RoboDK station: ur5_and_table_and_gripper.rdk

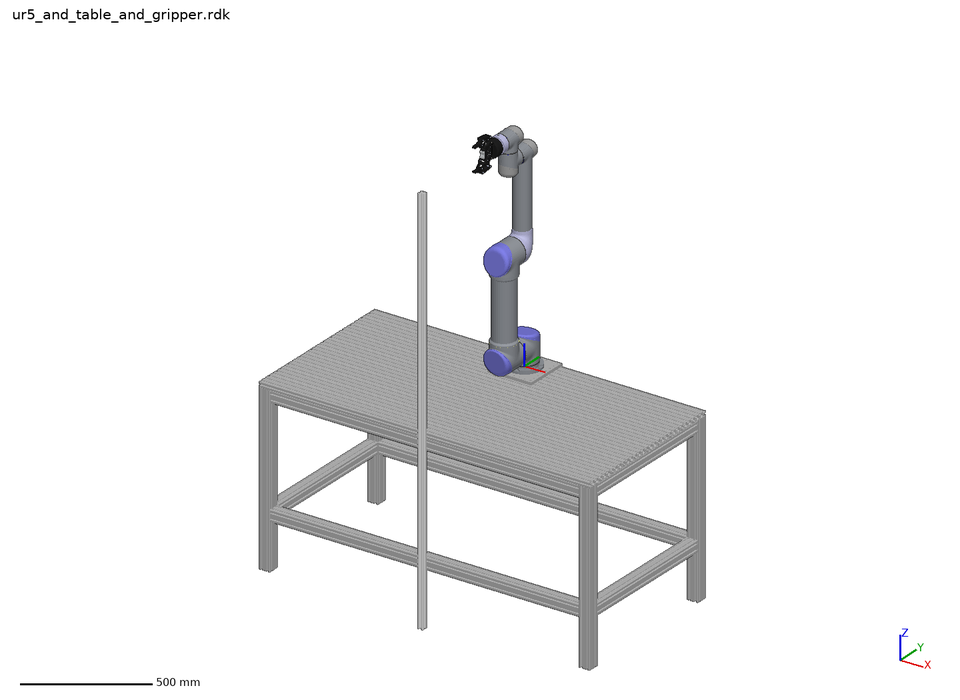
[picture v0: the station drawn from its stored meshes, robots at their saved joint values, targets as dots, program paths as lines]
Station ur5_and_table_and_gripper (saved by RoboDK 5.3.4). Poses are relative to the parent item; angles as X-Y-Z fixed-axis rotations.
  - frame UR5 Base at (0, 0, 0) mm
    - robot UR5: 6 axes, payload 5 kg, reach 850 mm, repeatability 0.1 mm, weight 18.4 kg
        modified DH rows (alpha deg, a mm, theta deg, d mm): 0, 0, 0, 89.2; 90, 0, 180, 0; 0, 425, 0, 0; 0, 392.43, 0, 109; -90, 0, 0, 93.65; 90, 0, 180, 82
        joint limits [-360, -360, -360, -360, -360, -360] to [360, 360, 360, 360, 360, 360]; home [0, -90, 90, 0, 90, 0]; saved at [0, -90, 0, -90, 0, 0]
      - tool Gripper RobotiQ 85 Opened, TCP at (0, 0, 149.6) mm, size 147.4 x 146.8 x 75 mm
  - object table_base_setup at (0, 0, 0) mm, rotated rx 0 ry 0 rz -90 deg, size 1524 x 762 x 800.1 mm, geometry from table_base_setup.STEP
  - object 6ft_beam_table at (0, -675, 1000) mm, size 25.4 x 25.4 x 1828.8 mm, geometry from 6ft_beam_table.IGS
  - Python program Task1 (listed below)
  - Python program Task 2 (listed below)
  - Python program Task 3 (listed below)

--- Python program Task1 ---
# This macro shows an example of running a program on the robot using the Python API (online programming)
# More information about the RoboDK API appears here:
# https://robodk.com/doc/en/RoboDK-API.html
from robolink import *    # API to communicate with RoboDK
from robodk import *      # robodk robotics toolbox
# Any interaction with RoboDK must be done through RDK:
RDK = Robolink()
# Select a robot (a popup is displayed if more than one robot is available)
robot = RDK.ItemUserPick('Select a robot', ITEM_TYPE_ROBOT)
if not robot.Valid():
    raise Exception('No robot selected or available')
RUN_ON_ROBOT = False
# Important: by default, the run mode is RUNMODE_SIMULATE
# If the program is generated offline manually the runmode will be RUNMODE_MAKE_ROBOTPROG,
# Therefore, we should not run the program on the robot
if RDK.RunMode() != RUNMODE_SIMULATE:
    RUN_ON_ROBOT = False
if RUN_ON_ROBOT:

    # Connect to the robot using default IP
    success = robot.Connect() # Try to connect once
    status, status_msg = robot.ConnectedState()
    if status != ROBOTCOM_READY:
        # Stop if the connection did not succeed
        print(status_msg)
        raise Exception("Failed to connect: " + status_msg)
    # This will set to run the API programs on the robot and the simulator (online programming)
    RDK.setRunMode(RUNMODE_RUN_ROBOT)



# Get the current joint position of the robot
# (updates the position on the robot simulator)
joints_ref = robot.Joints()
# get the current position of the TCP with respect to the reference frame:
# (4x4 matrix representing position and orientation)
target_ref = robot.Pose()
pos_ref = target_ref.Pos()
# It is important to provide the reference frame and the tool frames when generating programs offline
# It is important to update the TCP on the robot mostly when using the driver
robot.setPoseFrame(robot.PoseFrame())
robot.setPoseTool(robot.PoseTool())
#robot.setZoneData(10) # Set the rounding parameter (Also known as: CNT, APO/C_DIS, ZoneData, Blending radius, cornering, ...)





#Header above is re-used from the file provided for the first lab, not sure if all of it is needed but it can't hurt

#Actual Task 1 RoboDK Python segment:

#run rq_open
robot.RunCodeCustom('rq_open()',INSTRUCTION_CALL_PROGRAM)
robot.RunCodeCustom('sleep(5)',INSTRUCTION_CALL_PROGRAM)
#run rq_close
robot.RunCodeCustom('rq_close()',INSTRUCTION_CALL_PROGRAM)
robot.RunCodeCustom('sleep(5)',INSTRUCTION_CALL_PROGRAM)
#run rq_open_and_wait()
robot.RunCodeCustom('rq_open_and_wait()',INSTRUCTION_CALL_PROGRAM)
robot.RunCodeCustom('sleep(5)',INSTRUCTION_CALL_PROGRAM)
#run rq_close_and_wait()
robot.RunCodeCustom('rq_close_and_wait()',INSTRUCTION_CALL_PROGRAM)
robot.RunCodeCustom('sleep(5)',INSTRUCTION_CALL_PROGRAM)

#done

--- Python program Task 2 ---
# This macro shows an example of running a program on the robot using the Python API (online programming)
# More information about the RoboDK API appears here:
# https://robodk.com/doc/en/RoboDK-API.html
from robolink import *    # API to communicate with RoboDK
from robodk import *      # robodk robotics toolbox
# Any interaction with RoboDK must be done through RDK:
RDK = Robolink()
# Select a robot (a popup is displayed if more than one robot is available)
robot = RDK.ItemUserPick('Select a robot', ITEM_TYPE_ROBOT)
if not robot.Valid():
    raise Exception('No robot selected or available')
RUN_ON_ROBOT = False
# Important: by default, the run mode is RUNMODE_SIMULATE
# If the program is generated offline manually the runmode will be RUNMODE_MAKE_ROBOTPROG,
# Therefore, we should not run the program on the robot
if RDK.RunMode() != RUNMODE_SIMULATE:
    RUN_ON_ROBOT = False
if RUN_ON_ROBOT:

    # Connect to the robot using default IP
    success = robot.Connect() # Try to connect once
    status, status_msg = robot.ConnectedState()
    if status != ROBOTCOM_READY:
        # Stop if the connection did not succeed
        print(status_msg)
        raise Exception("Failed to connect: " + status_msg)
    # This will set to run the API programs on the robot and the simulator (online programming)
    RDK.setRunMode(RUNMODE_RUN_ROBOT)

# Get the current joint position of the robot
# (updates the position on the robot simulator)
joints_ref = robot.Joints()
# get the current position of the TCP with respect to the reference frame:
# (4x4 matrix representing position and orientation)
target_ref = robot.Pose()
pos_ref = target_ref.Pos()
# It is important to provide the reference frame and the tool frames when generating programs offline
# It is important to update the TCP on the robot mostly when using the driver
robot.setPoseFrame(robot.PoseFrame())
robot.setPoseTool(robot.PoseTool())
#robot.setZoneData(10) # Set the rounding parameter (Also known as: CNT, APO/C_DIS, ZoneData, Blending radius, cornering, ...)
robot.setSpeed(200) # Set linear speed in mm/s

# Setting Pose 1, Pose 2, and Pose 3 from the Lab Manual
# We enter our xyzrpw (X, Y, Z, RX, RY, RZ) into the function xyzrpw_2_pose()
# to convert out position and euler angles to a 4x4 pose matrix
# Start at the home position
home = [0, -90, 0, -90, 0, 0]

#Start Task 2 Program:

#since we are free driving to the position of the load cell, we don't have to move the robot pose at all, we will manually
#enter in the orientation ("RX:0","RY:3.146","RZ:0")

#initialize all the speeds and forces
forces = [0,1,50,100,127,128,150,200,255]
speeds = [25,50,75,105,150,200,250]

#initialize the gripper as open before starting the cycle:
robot.RunCodeCustom('rq_open_and_wait()',INSTRUCTION_CALL_PROGRAM)

#main for loop
for force in range (0,8):
    #Set force for next 7 iter
    robot.RunCodeCustom('rq_set_force(%i)' %forces[force],INSTRUCTION_CALL_PROGRAM)
    for speed in range (0,6):
        #Set speed for iter
        robot.RunCodeCustom('rq_set_speed(%i)' %speeds[speed],INSTRUCTION_CALL_PROGRAM)
        #Grasp
        robot.RunCodeCustom('rq_close_and_wait()',INSTRUCTION_CALL_PROGRAM)
        #Wait 2 seconds
        robot.RunCodeCustom('sleep(2)',INSTRUCTION_CALL_PROGRAM)
        #Fully open to be ready for next speed
        robot.RunCodeCustom('rq_open_and_wait()',INSTRUCTION_CALL_PROGRAM)

#Task 2 Complete

--- Python program Task 3 ---
# Type help("robolink") or help("robodk") for more information
# Press F5 to run the script
# Documentation: https://robodk.com/doc/en/RoboDK-API.html
# Reference:     https://robodk.com/doc/en/PythonAPI/index.html
# Note: It is not required to keep a copy of this file, your python script is saved with the station
from robolink import *    # RoboDK API
from robodk import *      # Robot toolbox
RDK = Robolink()

# Notify user:
print('To edit this program:\nright click on the Python program, then, select "Edit Python script"')

# Program example:
item = RDK.Item('base')
if item.Valid():
    print('Item selected: ' + item.Name())
    print('Item posistion: ' + repr(item.Pose()))

print('Items in the station:')
itemlist = RDK.ItemList()
print(itemlist)

raise Exception('Program not edited.')
